Staubli VAL3: deleteMove.pgx

public program deleteMove()
begin
  resetMotion()
  pDest=here(tActive,frActive)
end
